// TIA Portal V20 export
FUNCTION "FC_PositionCheck" : Void   // FC30, SCL
{ S7_Optimized_Access := 'TRUE' }
// stored: SetENOAutomatically false
   VAR_INPUT
      iAxisCurrentPos : LReal;
      iAxisTargetPos : LReal;
      iTolMin : Real;
      iTolMax : Real;
   END_VAR
   VAR_OUTPUT
      iInPos : Bool;
   END_VAR
BEGIN
   REGION Description header 
       //==================================================================================
       // POSALUX Swiss SA / (C) Copyright 2025
       //----------------------------------------------------------------------------------
       // Title: FC_PositionCheck
       // Comment/Function: 
       // Author: Fabien WALDT
       // Engineering: TIA Portal v17
       //----------------------------------------------------------------------------------
       // Change log table:
       // Version  | Date     | Expert in charge | Changes applied
       // ---------|----------|------------------|-----------------------------------------
       // 00.00.01 | 20250527 | WFA              | First released version
       // =================================================================================
   END_REGION

   REGION Check In Position
       IF #iAxisCurrentPos <= #iAxisTargetPos + #iTolMax
           AND #iAxisCurrentPos >= #iAxisTargetPos - #iTolMin THEN
           #iInPos := TRUE;
       ELSE
           #iInPos := FALSE;
       END_IF;
   END_REGION
END_FUNCTION
